REGION Network 130: FIXTURE IN UNIT 02 STATION 0 ANY CALIBRATION MISSING
   RUNG wire#powerrail
      Contact( "M_ONE" )
      wire#w1
      Contact( "DB4000_FIX_TABLE_POSITIONS".UNIT_02.FIXTURE_1.IN_LOAD_UNLOAD_STATION_1 )
      Contact( "DB7240_HARDWARE_SOFTWARE_ENABLE_DISABLE".DISABLE_FIXTURE.SW_UNIT_02_FIX_1_4_ENABLED )
      wire#w2
      Contact( "DB16010_MEASURE_SENSORS_CALIBRATION_STATUS".U02_STA2_MEAS.FIXTURE_1_MISSING )
      Contact( "DB7255_UNIT_02_STA_2_MEAS_ENABLE_DISABLE".ENABLED )
      wire#w3
      Coil( "DB2440_GLOBAL_DATA".GLOBAL_DATA.FIX_IN_UNIT_02_STA_0_ANY_CALIBRATION_MISS )
   END_RUNG
   RUNG wire#w2
      Contact( "DB16010_MEASURE_SENSORS_CALIBRATION_STATUS".U02_STA3_MEAS.FIXTURE_1_MISSING )
      Contact( "DB7256_UNIT_02_STA_3_MEAS_ENABLE_DISABLE".ENABLED )
   END_RUNG wire#w3
   RUNG wire#w1
      Contact( "DB4000_FIX_TABLE_POSITIONS".UNIT_02.FIXTURE_2.IN_LOAD_UNLOAD_STATION_1 )
      Contact( "DB7240_HARDWARE_SOFTWARE_ENABLE_DISABLE".DISABLE_FIXTURE.SW_UNIT_02_FIX_2_3_ENABLED )
      wire#w4
      Contact( "DB16010_MEASURE_SENSORS_CALIBRATION_STATUS".U02_STA2_MEAS.FIXTURE_2_MISSING )
      Contact( "DB7255_UNIT_02_STA_2_MEAS_ENABLE_DISABLE".ENABLED )
   END_RUNG wire#w3
   RUNG wire#w4
      Contact( "DB16010_MEASURE_SENSORS_CALIBRATION_STATUS".U02_STA3_MEAS.FIXTURE_2_MISSING )
      Contact( "DB7256_UNIT_02_STA_3_MEAS_ENABLE_DISABLE".ENABLED )
   END_RUNG wire#w3
   RUNG wire#w1
      Contact( "DB4000_FIX_TABLE_POSITIONS".UNIT_02.FIXTURE_3.IN_LOAD_UNLOAD_STATION_1 )
      Contact( "DB7240_HARDWARE_SOFTWARE_ENABLE_DISABLE".DISABLE_FIXTURE.SW_UNIT_02_FIX_2_3_ENABLED )
      wire#w5
      Contact( "DB16010_MEASURE_SENSORS_CALIBRATION_STATUS".U02_STA2_MEAS.FIXTURE_3_MISSING )
      Contact( "DB7255_UNIT_02_STA_2_MEAS_ENABLE_DISABLE".ENABLED )
   END_RUNG wire#w3
   RUNG wire#w5
      Contact( "DB16010_MEASURE_SENSORS_CALIBRATION_STATUS".U02_STA3_MEAS.FIXTURE_3_MISSING )
      Contact( "DB7256_UNIT_02_STA_3_MEAS_ENABLE_DISABLE".ENABLED )
   END_RUNG wire#w3
   RUNG wire#w1
      Contact( "DB4000_FIX_TABLE_POSITIONS".UNIT_02.FIXTURE_4.IN_LOAD_UNLOAD_STATION_1 )
      Contact( "DB7240_HARDWARE_SOFTWARE_ENABLE_DISABLE".DISABLE_FIXTURE.SW_UNIT_02_FIX_1_4_ENABLED )
      wire#w6
      Contact( "DB16010_MEASURE_SENSORS_CALIBRATION_STATUS".U02_STA2_MEAS.FIXTURE_4_MISSING )
      Contact( "DB7255_UNIT_02_STA_2_MEAS_ENABLE_DISABLE".ENABLED )
   END_RUNG wire#w3
   RUNG wire#w6
      Contact( "DB16010_MEASURE_SENSORS_CALIBRATION_STATUS".U02_STA3_MEAS.FIXTURE_4_MISSING )
      Contact( "DB7256_UNIT_02_STA_3_MEAS_ENABLE_DISABLE".ENABLED )
   END_RUNG wire#w3
   // the same network as SCL:
   "DB2440_GLOBAL_DATA".GLOBAL_DATA.FIX_IN_UNIT_02_STA_0_ANY_CALIBRATION_MISS := "M_ONE" AND (("DB4000_FIX_TABLE_POSITIONS".UNIT_02.FIXTURE_1.IN_LOAD_UNLOAD_STATION_1 AND "DB7240_HARDWARE_SOFTWARE_ENABLE_DISABLE".DISABLE_FIXTURE.SW_UNIT_02_FIX_1_4_ENABLED AND (("DB16010_MEASURE_SENSORS_CALIBRATION_STATUS".U02_STA2_MEAS.FIXTURE_1_MISSING AND "DB7255_UNIT_02_STA_2_MEAS_ENABLE_DISABLE".ENABLED) OR ("DB16010_MEASURE_SENSORS_CALIBRATION_STATUS".U02_STA3_MEAS.FIXTURE_1_MISSING AND "DB7256_UNIT_02_STA_3_MEAS_ENABLE_DISABLE".ENABLED))) OR ("DB4000_FIX_TABLE_POSITIONS".UNIT_02.FIXTURE_2.IN_LOAD_UNLOAD_STATION_1 AND "DB7240_HARDWARE_SOFTWARE_ENABLE_DISABLE".DISABLE_FIXTURE.SW_UNIT_02_FIX_2_3_ENABLED AND (("DB16010_MEASURE_SENSORS_CALIBRATION_STATUS".U02_STA2_MEAS.FIXTURE_2_MISSING AND "DB7255_UNIT_02_STA_2_MEAS_ENABLE_DISABLE".ENABLED) OR ("DB16010_MEASURE_SENSORS_CALIBRATION_STATUS".U02_STA3_MEAS.FIXTURE_2_MISSING AND "DB7256_UNIT_02_STA_3_MEAS_ENABLE_DISABLE".ENABLED))) OR ("DB4000_FIX_TABLE_POSITIONS".UNIT_02.FIXTURE_3.IN_LOAD_UNLOAD_STATION_1 AND "DB7240_HARDWARE_SOFTWARE_ENABLE_DISABLE".DISABLE_FIXTURE.SW_UNIT_02_FIX_2_3_ENABLED AND (("DB16010_MEASURE_SENSORS_CALIBRATION_STATUS".U02_STA2_MEAS.FIXTURE_3_MISSING AND "DB7255_UNIT_02_STA_2_MEAS_ENABLE_DISABLE".ENABLED) OR ("DB16010_MEASURE_SENSORS_CALIBRATION_STATUS".U02_STA3_MEAS.FIXTURE_3_MISSING AND "DB7256_UNIT_02_STA_3_MEAS_ENABLE_DISABLE".ENABLED))) OR ("DB4000_FIX_TABLE_POSITIONS".UNIT_02.FIXTURE_4.IN_LOAD_UNLOAD_STATION_1 AND "DB7240_HARDWARE_SOFTWARE_ENABLE_DISABLE".DISABLE_FIXTURE.SW_UNIT_02_FIX_1_4_ENABLED AND (("DB16010_MEASURE_SENSORS_CALIBRATION_STATUS".U02_STA2_MEAS.FIXTURE_4_MISSING AND "DB7255_UNIT_02_STA_2_MEAS_ENABLE_DISABLE".ENABLED) OR ("DB16010_MEASURE_SENSORS_CALIBRATION_STATUS".U02_STA3_MEAS.FIXTURE_4_MISSING AND "DB7256_UNIT_02_STA_3_MEAS_ENABLE_DISABLE".ENABLED))));
END_REGION

REGION Network 131: UNIT 01 ANY FIXTURE CALIBRATION MISSING
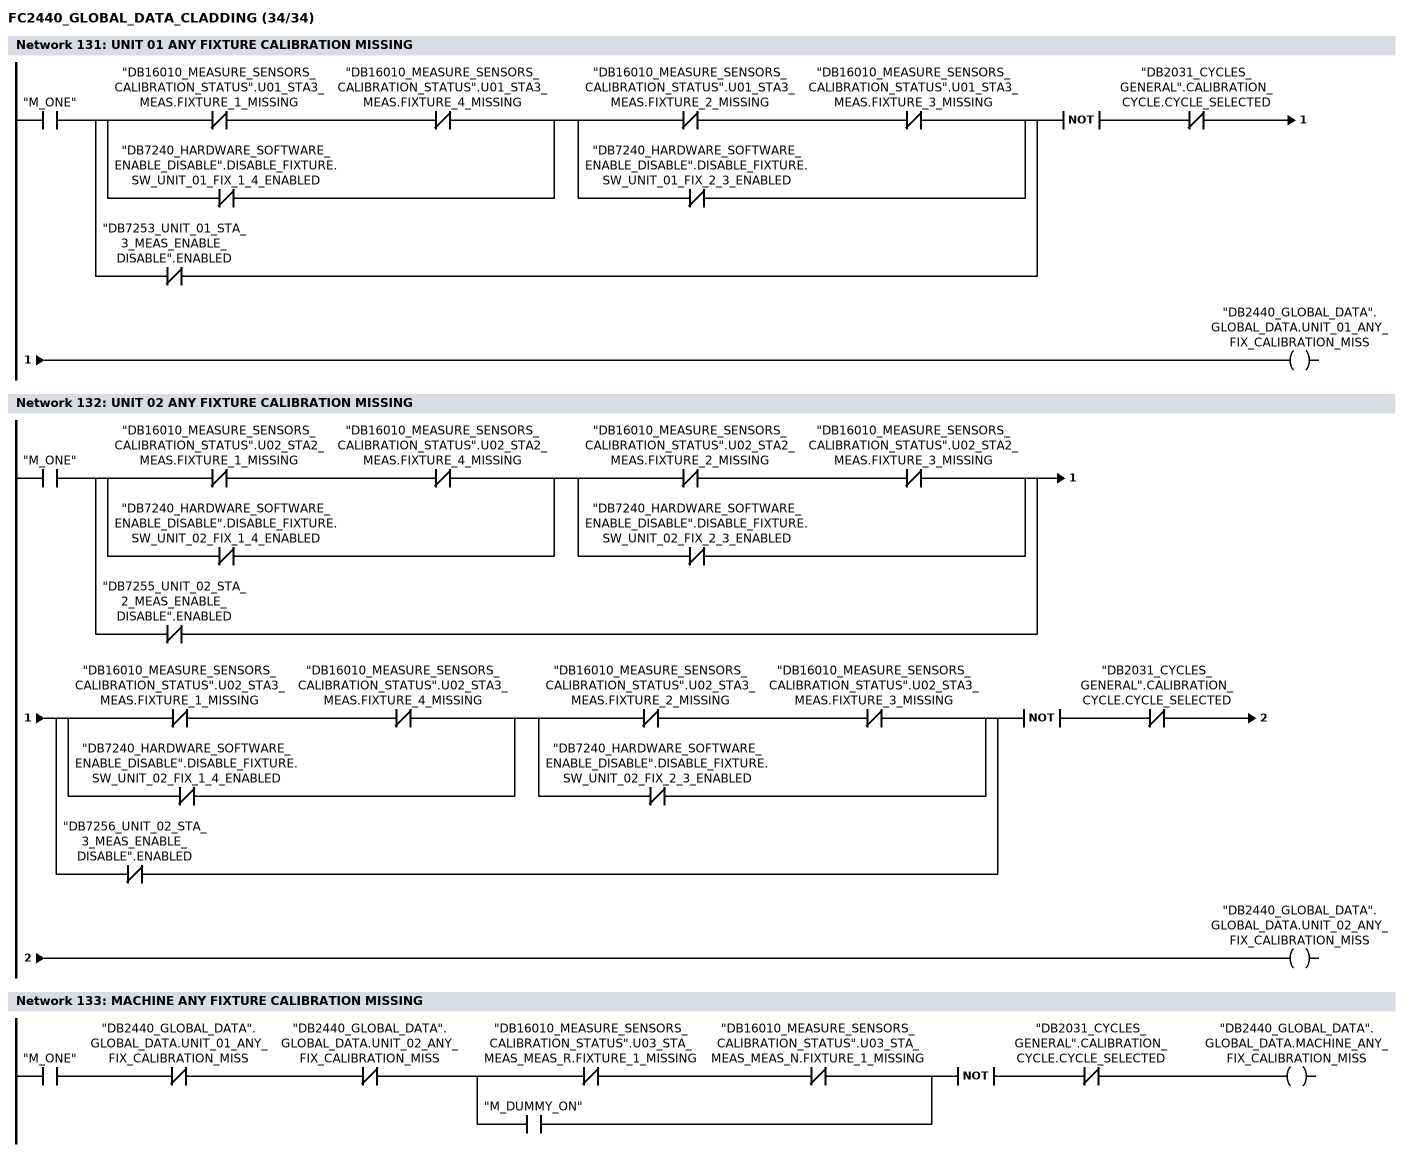
   RUNG wire#powerrail
      Contact( "M_ONE" )
      wire#w1
      I_Contact( "DB16010_MEASURE_SENSORS_CALIBRATION_STATUS".U01_STA3_MEAS.FIXTURE_1_MISSING )
      I_Contact( "DB16010_MEASURE_SENSORS_CALIBRATION_STATUS".U01_STA3_MEAS.FIXTURE_4_MISSING )
      wire#w2
      I_Contact( "DB16010_MEASURE_SENSORS_CALIBRATION_STATUS".U01_STA3_MEAS.FIXTURE_2_MISSING )
      I_Contact( "DB16010_MEASURE_SENSORS_CALIBRATION_STATUS".U01_STA3_MEAS.FIXTURE_3_MISSING )
      wire#w3
      Not()
      I_Contact( "DB2031_CYCLES_GENERAL".CALIBRATION_CYCLE.CYCLE_SELECTED )
      Coil( "DB2440_GLOBAL_DATA".GLOBAL_DATA.UNIT_01_ANY_FIX_CALIBRATION_MISS )
   END_RUNG
   RUNG wire#w1
      I_Contact( "DB7240_HARDWARE_SOFTWARE_ENABLE_DISABLE".DISABLE_FIXTURE.SW_UNIT_01_FIX_1_4_ENABLED )
   END_RUNG wire#w2
   RUNG wire#w2
      I_Contact( "DB7240_HARDWARE_SOFTWARE_ENABLE_DISABLE".DISABLE_FIXTURE.SW_UNIT_01_FIX_2_3_ENABLED )
   END_RUNG wire#w3
   RUNG wire#w1
      I_Contact( "DB7253_UNIT_01_STA_3_MEAS_ENABLE_DISABLE".ENABLED )
   END_RUNG wire#w3
   // the same network as SCL:
   "DB2440_GLOBAL_DATA".GLOBAL_DATA.UNIT_01_ANY_FIX_CALIBRATION_MISS := NOT ("M_ONE" AND ((((NOT "DB16010_MEASURE_SENSORS_CALIBRATION_STATUS".U01_STA3_MEAS.FIXTURE_1_MISSING AND NOT "DB16010_MEASURE_SENSORS_CALIBRATION_STATUS".U01_STA3_MEAS.FIXTURE_4_MISSING) OR NOT "DB7240_HARDWARE_SOFTWARE_ENABLE_DISABLE".DISABLE_FIXTURE.SW_UNIT_01_FIX_1_4_ENABLED) AND ((NOT "DB16010_MEASURE_SENSORS_CALIBRATION_STATUS".U01_STA3_MEAS.FIXTURE_2_MISSING AND NOT "DB16010_MEASURE_SENSORS_CALIBRATION_STATUS".U01_STA3_MEAS.FIXTURE_3_MISSING) OR NOT "DB7240_HARDWARE_SOFTWARE_ENABLE_DISABLE".DISABLE_FIXTURE.SW_UNIT_01_FIX_2_3_ENABLED)) OR NOT "DB7253_UNIT_01_STA_3_MEAS_ENABLE_DISABLE".ENABLED)) AND NOT "DB2031_CYCLES_GENERAL".CALIBRATION_CYCLE.CYCLE_SELECTED;
END_REGION

REGION Network 132: UNIT 02 ANY FIXTURE CALIBRATION MISSING
   RUNG wire#powerrail
      Contact( "M_ONE" )
      wire#w1
      I_Contact( "DB16010_MEASURE_SENSORS_CALIBRATION_STATUS".U02_STA2_MEAS.FIXTURE_1_MISSING )
      I_Contact( "DB16010_MEASURE_SENSORS_CALIBRATION_STATUS".U02_STA2_MEAS.FIXTURE_4_MISSING )
      wire#w2
      I_Contact( "DB16010_MEASURE_SENSORS_CALIBRATION_STATUS".U02_STA2_MEAS.FIXTURE_2_MISSING )
      I_Contact( "DB16010_MEASURE_SENSORS_CALIBRATION_STATUS".U02_STA2_MEAS.FIXTURE_3_MISSING )
      wire#w3
      I_Contact( "DB16010_MEASURE_SENSORS_CALIBRATION_STATUS".U02_STA3_MEAS.FIXTURE_1_MISSING )
      I_Contact( "DB16010_MEASURE_SENSORS_CALIBRATION_STATUS".U02_STA3_MEAS.FIXTURE_4_MISSING )
      wire#w4
      I_Contact( "DB16010_MEASURE_SENSORS_CALIBRATION_STATUS".U02_STA3_MEAS.FIXTURE_2_MISSING )
      I_Contact( "DB16010_MEASURE_SENSORS_CALIBRATION_STATUS".U02_STA3_MEAS.FIXTURE_3_MISSING )
      wire#w5
      Not()
      I_Contact( "DB2031_CYCLES_GENERAL".CALIBRATION_CYCLE.CYCLE_SELECTED )
      Coil( "DB2440_GLOBAL_DATA".GLOBAL_DATA.UNIT_02_ANY_FIX_CALIBRATION_MISS )
   END_RUNG
   RUNG wire#w1
      I_Contact( "DB7240_HARDWARE_SOFTWARE_ENABLE_DISABLE".DISABLE_FIXTURE.SW_UNIT_02_FIX_1_4_ENABLED )
   END_RUNG wire#w2
   RUNG wire#w2
      I_Contact( "DB7240_HARDWARE_SOFTWARE_ENABLE_DISABLE".DISABLE_FIXTURE.SW_UNIT_02_FIX_2_3_ENABLED )
   END_RUNG wire#w3
   RUNG wire#w1
      I_Contact( "DB7255_UNIT_02_STA_2_MEAS_ENABLE_DISABLE".ENABLED )
   END_RUNG wire#w3
   RUNG wire#w3
      I_Contact( "DB7240_HARDWARE_SOFTWARE_ENABLE_DISABLE".DISABLE_FIXTURE.SW_UNIT_02_FIX_1_4_ENABLED )
   END_RUNG wire#w4
   RUNG wire#w4
      I_Contact( "DB7240_HARDWARE_SOFTWARE_ENABLE_DISABLE".DISABLE_FIXTURE.SW_UNIT_02_FIX_2_3_ENABLED )
   END_RUNG wire#w5
   RUNG wire#w3
      I_Contact( "DB7256_UNIT_02_STA_3_MEAS_ENABLE_DISABLE".ENABLED )
   END_RUNG wire#w5
   // the same network as SCL:
   "DB2440_GLOBAL_DATA".GLOBAL_DATA.UNIT_02_ANY_FIX_CALIBRATION_MISS := NOT ("M_ONE" AND ((((NOT "DB16010_MEASURE_SENSORS_CALIBRATION_STATUS".U02_STA2_MEAS.FIXTURE_1_MISSING AND NOT "DB16010_MEASURE_SENSORS_CALIBRATION_STATUS".U02_STA2_MEAS.FIXTURE_4_MISSING) OR NOT "DB7240_HARDWARE_SOFTWARE_ENABLE_DISABLE".DISABLE_FIXTURE.SW_UNIT_02_FIX_1_4_ENABLED) AND ((NOT "DB16010_MEASURE_SENSORS_CALIBRATION_STATUS".U02_STA2_MEAS.FIXTURE_2_MISSING AND NOT "DB16010_MEASURE_SENSORS_CALIBRATION_STATUS".U02_STA2_MEAS.FIXTURE_3_MISSING) OR NOT "DB7240_HARDWARE_SOFTWARE_ENABLE_DISABLE".DISABLE_FIXTURE.SW_UNIT_02_FIX_2_3_ENABLED)) OR NOT "DB7255_UNIT_02_STA_2_MEAS_ENABLE_DISABLE".ENABLED) AND ((((NOT "DB16010_MEASURE_SENSORS_CALIBRATION_STATUS".U02_STA3_MEAS.FIXTURE_1_MISSING AND NOT "DB16010_MEASURE_SENSORS_CALIBRATION_STATUS".U02_STA3_MEAS.FIXTURE_4_MISSING) OR NOT "DB7240_HARDWARE_SOFTWARE_ENABLE_DISABLE".DISABLE_FIXTURE.SW_UNIT_02_FIX_1_4_ENABLED) AND ((NOT "DB16010_MEASURE_SENSORS_CALIBRATION_STATUS".U02_STA3_MEAS.FIXTURE_2_MISSING AND NOT "DB16010_MEASURE_SENSORS_CALIBRATION_STATUS".U02_STA3_MEAS.FIXTURE_3_MISSING) OR NOT "DB7240_HARDWARE_SOFTWARE_ENABLE_DISABLE".DISABLE_FIXTURE.SW_UNIT_02_FIX_2_3_ENABLED)) OR NOT "DB7256_UNIT_02_STA_3_MEAS_ENABLE_DISABLE".ENABLED)) AND NOT "DB2031_CYCLES_GENERAL".CALIBRATION_CYCLE.CYCLE_SELECTED;
END_REGION

REGION Network 133: MACHINE ANY FIXTURE CALIBRATION MISSING
   RUNG wire#powerrail
      Contact( "M_ONE" )
      I_Contact( "DB2440_GLOBAL_DATA".GLOBAL_DATA.UNIT_01_ANY_FIX_CALIBRATION_MISS )
      I_Contact( "DB2440_GLOBAL_DATA".GLOBAL_DATA.UNIT_02_ANY_FIX_CALIBRATION_MISS )
      wire#w1
      I_Contact( "DB16010_MEASURE_SENSORS_CALIBRATION_STATUS".U03_STA_MEAS_MEAS_R.FIXTURE_1_MISSING )
      I_Contact( "DB16010_MEASURE_SENSORS_CALIBRATION_STATUS".U03_STA_MEAS_MEAS_N.FIXTURE_1_MISSING )
      wire#w2
      Not()
      I_Contact( "DB2031_CYCLES_GENERAL".CALIBRATION_CYCLE.CYCLE_SELECTED )
      Coil( "DB2440_GLOBAL_DATA".GLOBAL_DATA.MACHINE_ANY_FIX_CALIBRATION_MISS )
   END_RUNG
   RUNG wire#w1
      Contact( "M_DUMMY_ON" )
   END_RUNG wire#w2
   // the same network as SCL:
   "DB2440_GLOBAL_DATA".GLOBAL_DATA.MACHINE_ANY_FIX_CALIBRATION_MISS := NOT ("M_ONE" AND NOT "DB2440_GLOBAL_DATA".GLOBAL_DATA.UNIT_01_ANY_FIX_CALIBRATION_MISS AND NOT "DB2440_GLOBAL_DATA".GLOBAL_DATA.UNIT_02_ANY_FIX_CALIBRATION_MISS AND ((NOT "DB16010_MEASURE_SENSORS_CALIBRATION_STATUS".U03_STA_MEAS_MEAS_R.FIXTURE_1_MISSING AND NOT "DB16010_MEASURE_SENSORS_CALIBRATION_STATUS".U03_STA_MEAS_MEAS_N.FIXTURE_1_MISSING) OR "M_DUMMY_ON")) AND NOT "DB2031_CYCLES_GENERAL".CALIBRATION_CYCLE.CYCLE_SELECTED;
END_REGION
END_FUNCTION
